(* IEC 61131-3 sources: statemachine/src/StatePattern, 2 files *)

(* ---- BaseState.st ---- *)
USING Simatic.Ax.StatePattern;
NAMESPACE Simatic.Ax.StatePattern
    CLASS StateBase IMPLEMENTS IState
        VAR
            _nextState : IState;
            _nextStateTimeout : IState;
        END_VAR

        METHOD PUBLIC Config
            VAR_INPUT
                nextState : IState;
                nextStateTimeout : IState;
            END_VAR
            _nextState := nextState;
            _nextStateTimeout := nextStateTimeout;
        END_METHOD

        METHOD PUBLIC OnTimeout
            VAR_INPUT
                context : REF_TO StateContext;
            END_VAR
            ;
        END_METHOD

        METHOD PUBLIC Execute
            VAR_INPUT
                context : REF_TO StateContext;
            END_VAR
            ;
        END_METHOD

        METHOD PUBLIC OnEntry
            VAR_INPUT
                context : REF_TO StateContext;
            END_VAR;
        END_METHOD

        METHOD PUBLIC OnExit
            VAR_INPUT
                context : REF_TO StateContext;
            END_VAR;
        END_METHOD

    END_CLASS
END_NAMESPACE

(* ---- StateContext.st ---- *)
USING System.Timer;

NAMESPACE Simatic.Ax.StatePattern
    CLASS PUBLIC StateContext
        VAR PUBLIC

        END_VAR
        VAR
            _count : INT;
            _state : IState;
            _ton : OnDelay;
            _first : BOOL := TRUE;
            _status : StateStatus;
        END_VAR

        METHOD PUBLIC InitialState : BOOL
            VAR_INPUT
                newState : IState;
                timeout : TIME;
                reset : BOOL := FALSE;
            END_VAR

            IF (newState <> NULL) THEN
                IF (_first OR reset) THEN
                    THIS.setState(newState := newState, timeout := timeout);
                    _first := FALSE;
                END_IF;
                InitialState := TRUE;
            ELSE
                InitialState := FALSE;
            END_IF;

        END_METHOD

        METHOD PUBLIC FINAL SetState
            VAR_INPUT
                newState : IState;
                timeout : TIME;
            END_VAR

            // before change state, call the on Entry method
            IF (_state <> NULL) THEN
                _state.OnExit(context := REF(THIS));
            END_IF;

            IF (newState <> NULL) THEN
                _state := newState;
                _status.isRunning := TRUE;

                // call the OnEntry method once
                _state.onEntry(context := REF(THIS));

                // run the Timeout if configured
                IF (timeout > T#0ms) THEN
                    _ton.duration := timeout;
                    _ton.signal := TRUE;
                END_IF;
                _state.Execute(context := REF(THIS));

            END_IF;
        END_METHOD

        METHOD PUBLIC FINAL Execute
            IF (_state = NULL) THEN
                RETURN;
            END_IF;
            _count := _count + 1;
            _ton();

            IF (_ton.output) THEN
                _ton.signal := FALSE;
                _ton();
                _status.remainingTime := _ton.elapsedTime;
                _state.OnTimeout(context := REF(THIS));
            END_IF;

            _state.Execute(context := REF(THIS));
        END_METHOD

    END_CLASS
END_NAMESPACE
